// TIA Portal V20 export
TYPE "type_emRelations_em7_cmStatus"
// stored: Access Published, Namespace Unit1
   STRUCT
      cmSepaClampDetectSensor { ExternalAccessible := 'False'; ExternalVisible := 'False'; ExternalWritable := 'False'} : "LBC_typeDigitalSignalControlNode";
      cmSepaGripperDetectSensor { ExternalAccessible := 'False'; ExternalVisible := 'False'; ExternalWritable := 'False'} : "LBC_typeDigitalSignalControlNode";
      cmJRWinderDetectSensor { ExternalAccessible := 'False'; ExternalVisible := 'False'; ExternalWritable := 'False'} : "LBC_typeDigitalSignalControlNode";
      cmSepaClampSafetyPinDetectSensor { ExternalAccessible := 'False'; ExternalVisible := 'False'; ExternalWritable := 'False'} : "LBC_typeDigitalSignalControlNode";
      cmSepaGripperSafetyPinDetectSensor { ExternalAccessible := 'False'; ExternalVisible := 'False'; ExternalWritable := 'False'} : "LBC_typeDigitalSignalControlNode";
      cmSepaClampnCutterAxisX { ExternalAccessible := 'False'; ExternalVisible := 'False'; ExternalWritable := 'False'} : "LBC_typeAxis64PosControlNode";
      cmSepaClampnCutterAxisZ { ExternalAccessible := 'False'; ExternalVisible := 'False'; ExternalWritable := 'False'} : "LBC_typeAxis64PosControlNode";
      cmSepaGripperAxisX { ExternalAccessible := 'False'; ExternalVisible := 'False'; ExternalWritable := 'False'} : "LBC_typeAxis64PosControlNode";
      cmSepaGripperAxisZ { ExternalAccessible := 'False'; ExternalVisible := 'False'; ExternalWritable := 'False'} : "LBC_typeAxis64PosControlNode";
      cmSepaGripperAxisC { ExternalAccessible := 'False'; ExternalVisible := 'False'; ExternalWritable := 'False'} : "LBC_typeAxis64PosControlNode";
      cmJRWinderRearAxisY { ExternalAccessible := 'False'; ExternalVisible := 'False'; ExternalWritable := 'False'} : "LBC_typeAxis64PosControlNode";
      cmJRWinderFrontAxisY { ExternalAccessible := 'False'; ExternalVisible := 'False'; ExternalWritable := 'False'} : "LBC_typeAxis64PosControlNode";
      cmJRWinderAxisB { ExternalAccessible := 'False'; ExternalVisible := 'False'; ExternalWritable := 'False'} : "LBC_typeAxis64PosControlNode";
      cmJRPusherAxisZ { ExternalAccessible := 'False'; ExternalVisible := 'False'; ExternalWritable := 'False'} : "LBC_typeAxis64PosControlNode";
      cmSepaCutterUpDown { ExternalAccessible := 'False'; ExternalVisible := 'False'; ExternalWritable := 'False'} : "LBC_typeTwoWayActuatorControlNode";
      cmSepaClampTopUpDown { ExternalAccessible := 'False'; ExternalVisible := 'False'; ExternalWritable := 'False'} : "LBC_typeTwoWayActuatorControlNode";
      cmSepaClampBottomUpDown { ExternalAccessible := 'False'; ExternalVisible := 'False'; ExternalWritable := 'False'} : "LBC_typeTwoWayActuatorControlNode";
      cmStackGripperOpenClose { ExternalAccessible := 'False'; ExternalVisible := 'False'; ExternalWritable := 'False'} : "LBC_typeTwoWayActuatorControlNode";
      cmStackGripperFwdBwd { ExternalAccessible := 'False'; ExternalVisible := 'False'; ExternalWritable := 'False'} : "LBC_typeTwoWayActuatorControlNode";
      cmJRWinderClampTopRearUpDown { ExternalAccessible := 'False'; ExternalVisible := 'False'; ExternalWritable := 'False'} : "LBC_typeTwoWayActuatorControlNode";
      cmJRWinderClampBtmRearUpDown { ExternalAccessible := 'False'; ExternalVisible := 'False'; ExternalWritable := 'False'} : "LBC_typeTwoWayActuatorControlNode";
      cmJRWinderClampTopFrontUpDown { ExternalAccessible := 'False'; ExternalVisible := 'False'; ExternalWritable := 'False'} : "LBC_typeTwoWayActuatorControlNode";
      cmJRWinderClampBtmFrontUpDown { ExternalAccessible := 'False'; ExternalVisible := 'False'; ExternalWritable := 'False'} : "LBC_typeTwoWayActuatorControlNode";
      cmPusherRollerFwdBwd { ExternalAccessible := 'False'; ExternalVisible := 'False'; ExternalWritable := 'False'} : "LBC_typeTwoWayActuatorControlNode";
      cmHotWireCutter { ExternalAccessible := 'False'; ExternalVisible := 'False'; ExternalWritable := 'False'} : "LER_typeHotWireCutterControlNode";
   END_STRUCT;
   // cmSepaClampnCutterAxisX.commandConfiguration.power.startMode := 1;
   // cmSepaClampnCutterAxisX.commandConfiguration.power.stopMode := 0;
   // cmSepaClampnCutterAxisX.commandConfiguration.power.syncMotionSimulation := FALSE;
   // cmSepaClampnCutterAxisX.commandConfiguration.power.syncMotionSimulationExtendedMode := -1;
   // cmSepaClampnCutterAxisX.commandConfiguration.jog.velocity := 0.0;
   // cmSepaClampnCutterAxisX.commandConfiguration.jog.acceleration := -1.0;
   // cmSepaClampnCutterAxisX.commandConfiguration.jog.deceleration := -1.0;
   // cmSepaClampnCutterAxisX.commandConfiguration.jog.jerk := -1.0;
   // cmSepaClampnCutterAxisX.commandConfiguration.jog.positionControlled := TRUE;
   // cmSepaClampnCutterAxisX.commandConfiguration.jog.increment := 0.0;
   // cmSepaClampnCutterAxisX.commandConfiguration.jog.mode := 0;
   // cmSepaClampnCutterAxisX.commandConfiguration.moveVelocity.velocity := 0.0;
   // cmSepaClampnCutterAxisX.commandConfiguration.moveVelocity.acceleration := -1.0;
   // cmSepaClampnCutterAxisX.commandConfiguration.moveVelocity.deceleration := -1.0;
   // cmSepaClampnCutterAxisX.commandConfiguration.moveVelocity.jerk := -1.0;
   // cmSepaClampnCutterAxisX.commandConfiguration.moveVelocity.direction := 0;
   // cmSepaClampnCutterAxisX.commandConfiguration.moveVelocity.positionControlled := TRUE;
   // cmSepaClampnCutterAxisX.commandConfiguration.moveVelocity.velocityChangeOnTheFly := FALSE;
   // cmSepaClampnCutterAxisX.commandConfiguration.stop.deceleration := -1.0;
   // cmSepaClampnCutterAxisX.commandConfiguration.stop.jerk := -1.0;
   // cmSepaClampnCutterAxisX.commandConfiguration.stop.abortAcceleration := FALSE;
   // cmSepaClampnCutterAxisX.commandConfiguration.fastStop.deceleration := -1.0;
   // cmSepaClampnCutterAxisX.commandConfiguration.fastStop.jerk := -1.0;
   // cmSepaClampnCutterAxisX.commandConfiguration.fastStop.abortAcceleration := FALSE;
   // cmSepaClampnCutterAxisX.commandConfiguration.fastStop.replaceStopPossible := FALSE;
   // cmSepaClampnCutterAxisX.commandConfiguration.torqueLimiting.limit := -1.0;
   // cmSepaClampnCutterAxisX.commandConfiguration.torqueLimiting.mode := 0;
   // cmSepaClampnCutterAxisX.commandConfiguration.posRelative.distance := 0.0;
   // cmSepaClampnCutterAxisX.commandConfiguration.posRelative.velocity := -1.0;
   // cmSepaClampnCutterAxisX.commandConfiguration.posRelative.acceleration := -1.0;
   // cmSepaClampnCutterAxisX.commandConfiguration.posRelative.deceleration := -1.0;
   // cmSepaClampnCutterAxisX.commandConfiguration.posRelative.jerk := -1.0;
   // cmSepaClampnCutterAxisX.commandConfiguration.posRelative.direction := 0;
   // cmSepaClampnCutterAxisX.commandConfiguration.posAbsolute.position := 0.0;
   // cmSepaClampnCutterAxisX.commandConfiguration.posAbsolute.velocity := -1.0;
   // cmSepaClampnCutterAxisX.commandConfiguration.posAbsolute.acceleration := -1.0;
   // cmSepaClampnCutterAxisX.commandConfiguration.posAbsolute.deceleration := -1.0;
   // cmSepaClampnCutterAxisX.commandConfiguration.posAbsolute.jerk := -1.0;
   // cmSepaClampnCutterAxisX.commandConfiguration.posAbsolute.direction := 1;
   // cmSepaClampnCutterAxisX.commandConfiguration.posAbsolute.positionChangeOnTheFly := FALSE;
   // cmSepaClampnCutterAxisX.commandConfiguration.posAbsolute.velocityChangeOnTheFly := FALSE;
   // cmSepaClampnCutterAxisX.commandConfiguration.posSuperimposed.distance := 0.0;
   // cmSepaClampnCutterAxisX.commandConfiguration.posSuperimposed.velocityDiff := -1.0;
   // cmSepaClampnCutterAxisX.commandConfiguration.posSuperimposed.acceleration := -1.0;
   // cmSepaClampnCutterAxisX.commandConfiguration.posSuperimposed.deceleration := -1.0;
   // cmSepaClampnCutterAxisX.commandConfiguration.posSuperimposed.jerk := -1.0;
   // cmSepaClampnCutterAxisX.commandConfiguration.posSuperimposed.direction := 0;
   // cmSepaClampnCutterAxisX.commandConfiguration.haltSuperimposed.deceleration := -1.0;
   // cmSepaClampnCutterAxisX.commandConfiguration.haltSuperimposed.jerk := -1.0;
   // cmSepaClampnCutterAxisX.commandConfiguration.haltSuperimposed.abortAcceleration := FALSE;
   // cmSepaClampnCutterAxisX.commandConfiguration.gearInRelative.ratioNumerator := 1;
   // cmSepaClampnCutterAxisX.commandConfiguration.gearInRelative.ratioDenominator := 1;
   // cmSepaClampnCutterAxisX.commandConfiguration.gearInRelative.acceleration := -1.0;
   // cmSepaClampnCutterAxisX.commandConfiguration.gearInRelative.deceleration := -1.0;
   // cmSepaClampnCutterAxisX.commandConfiguration.gearInRelative.jerk := -1.0;
   // cmSepaClampnCutterAxisX.commandConfiguration.gearInRelative.ratioChangeOnTheFly := FALSE;
   // cmSepaClampnCutterAxisX.commandConfiguration.gearInAbsolute.ratioNumerator := 1;
   // cmSepaClampnCutterAxisX.commandConfiguration.gearInAbsolute.ratioDenominator := 1;
   // cmSepaClampnCutterAxisX.commandConfiguration.gearInAbsolute.masterSyncPosition := 0.0;
   // cmSepaClampnCutterAxisX.commandConfiguration.gearInAbsolute.slaveSyncPosition := 0.0;
   // cmSepaClampnCutterAxisX.commandConfiguration.gearInAbsolute.syncProfileReference := 1;
   // cmSepaClampnCutterAxisX.commandConfiguration.gearInAbsolute.masterStartDistance := 0.0;
   // cmSepaClampnCutterAxisX.commandConfiguration.gearInAbsolute.velocity := -1.0;
   // cmSepaClampnCutterAxisX.commandConfiguration.gearInAbsolute.acceleration := -1.0;
   // cmSepaClampnCutterAxisX.commandConfiguration.gearInAbsolute.deceleration := -1.0;
   // cmSepaClampnCutterAxisX.commandConfiguration.gearInAbsolute.jerk := -1.0;
   // cmSepaClampnCutterAxisX.commandConfiguration.gearInAbsolute.syncDirection := 1;
   // cmSepaClampnCutterAxisX.commandConfiguration.gearInAbsolute.ratioChangeOnTheFly := FALSE;
   // cmSepaClampnCutterAxisX.commandConfiguration.gearInVelocity.continuousUpdate := FALSE;
   // cmSepaClampnCutterAxisX.commandConfiguration.gearInVelocity.ratioNumerator := 1;
   // cmSepaClampnCutterAxisX.commandConfiguration.gearInVelocity.ratioDenominator := 1;
   // cmSepaClampnCutterAxisX.commandConfiguration.gearInVelocity.acceleration := -1.0;
   // cmSepaClampnCutterAxisX.commandConfiguration.gearInVelocity.deceleration := -1.0;
   // cmSepaClampnCutterAxisX.commandConfiguration.gearInVelocity.jerk := -1.0;
   // cmSepaClampnCutterAxisX.commandConfiguration.gearInVelocity.positionControlled := FALSE;
   // cmSepaClampnCutterAxisX.commandConfiguration.camIn.masterOffset := 0.0;
   // cmSepaClampnCutterAxisX.commandConfiguration.camIn.slaveOffset := 0.0;
   // cmSepaClampnCutterAxisX.commandConfiguration.camIn.masterScaling := 1.0;
   // cmSepaClampnCutterAxisX.commandConfiguration.camIn.slaveScaling := 1.0;
   // cmSepaClampnCutterAxisX.commandConfiguration.camIn.masterSyncPosition := 0.0;
   // cmSepaClampnCutterAxisX.commandConfiguration.camIn.syncProfileReference := 1;
   // cmSepaClampnCutterAxisX.commandConfiguration.camIn.masterStartDistance := 0.0;
   // cmSepaClampnCutterAxisX.commandConfiguration.camIn.velocity := -1.0;
   // cmSepaClampnCutterAxisX.commandConfiguration.camIn.acceleration := -1.0;
   // cmSepaClampnCutterAxisX.commandConfiguration.camIn.deceleration := -1.0;
   // cmSepaClampnCutterAxisX.commandConfiguration.camIn.jerk := -1.0;
   // cmSepaClampnCutterAxisX.commandConfiguration.camIn.applicationMode := 0;
   // cmSepaClampnCutterAxisX.commandConfiguration.camIn.syncDirection := 1;
   // cmSepaClampnCutterAxisX.commandConfiguration.gearOutCamOut.slavePosition := 0.0;
   // cmSepaClampnCutterAxisX.commandConfiguration.gearOutCamOut.syncProfileReference := 1;
   // cmSepaClampnCutterAxisX.commandConfiguration.gearOutCamOut.masterStopDistance := 0.0;
   // cmSepaClampnCutterAxisX.commandConfiguration.gearOutCamOut.deceleration := -1.0;
   // cmSepaClampnCutterAxisX.commandConfiguration.gearOutCamOut.jerk := -1.0;
   // cmSepaClampnCutterAxisX.commandConfiguration.gearOutCamOut.syncOutDirection := 3;
   // cmSepaClampnCutterAxisX.commandConfiguration.gearOutCamOut.gearOutCamOutMode := -1;
   // cmSepaClampnCutterAxisX.commandConfiguration.phasing.phaseShift := 0.0;
   // cmSepaClampnCutterAxisX.commandConfiguration.phasing.velocity := -1.0;
   // cmSepaClampnCutterAxisX.commandConfiguration.phasing.acceleration := -1.0;
   // cmSepaClampnCutterAxisX.commandConfiguration.phasing.deceleration := -1.0;
   // cmSepaClampnCutterAxisX.commandConfiguration.phasing.jerk := -1.0;
   // cmSepaClampnCutterAxisX.commandConfiguration.phasing.profileReference := 0;
   // cmSepaClampnCutterAxisX.commandConfiguration.phasing.phasingDistance := 0.0;
   // cmSepaClampnCutterAxisX.commandConfiguration.phasing.startPosition := 0.0;
   // cmSepaClampnCutterAxisX.commandConfiguration.phasing.direction := 3;
   // cmSepaClampnCutterAxisX.commandConfiguration.phasing.phaseAbsolute := TRUE;
   // cmSepaClampnCutterAxisX.commandConfiguration.phasing.phaseShiftChangeOnTheFly := FALSE;
   // cmSepaClampnCutterAxisX.commandConfiguration.offset.offset := 0.0;
   // cmSepaClampnCutterAxisX.commandConfiguration.offset.profileReference := 1;
   // cmSepaClampnCutterAxisX.commandConfiguration.offset.offsetDistance := 0.0;
   // cmSepaClampnCutterAxisX.commandConfiguration.offset.startPosition := 0.0;
   // cmSepaClampnCutterAxisX.commandConfiguration.offset.direction := 3;
   // cmSepaClampnCutterAxisX.commandConfiguration.offset.offsetAbsolute := TRUE;
   // cmSepaClampnCutterAxisX.commandConfiguration.offset.offsetChangeOnTheFly := FALSE;
   // cmSepaClampnCutterAxisZ.commandConfiguration.generalSettings.stopOnError := TRUE;
   // cmSepaClampnCutterAxisZ.commandConfiguration.generalSettings.resetWithRestart := FALSE;
   // cmSepaClampnCutterAxisZ.commandConfiguration.generalSettings.abortWaitingSyncCmd := TRUE;
   // cmSepaClampnCutterAxisZ.commandConfiguration.power.startMode := 1;
   // cmSepaClampnCutterAxisZ.commandConfiguration.power.stopMode := 0;
   // cmSepaClampnCutterAxisZ.commandConfiguration.power.syncMotionSimulation := FALSE;
   // cmSepaClampnCutterAxisZ.commandConfiguration.power.syncMotionSimulationExtendedMode := -1;
   // cmSepaClampnCutterAxisZ.commandConfiguration.jog.velocity := 0.0;
   // cmSepaClampnCutterAxisZ.commandConfiguration.jog.acceleration := -1.0;
   // cmSepaClampnCutterAxisZ.commandConfiguration.jog.deceleration := -1.0;
   // cmSepaClampnCutterAxisZ.commandConfiguration.jog.jerk := -1.0;
   // cmSepaClampnCutterAxisZ.commandConfiguration.jog.positionControlled := TRUE;
   // cmSepaClampnCutterAxisZ.commandConfiguration.jog.increment := 0.0;
   // cmSepaClampnCutterAxisZ.commandConfiguration.jog.mode := 0;
   // cmSepaClampnCutterAxisZ.commandConfiguration.moveVelocity.velocity := 0.0;
   // cmSepaClampnCutterAxisZ.commandConfiguration.moveVelocity.acceleration := -1.0;
   // cmSepaClampnCutterAxisZ.commandConfiguration.moveVelocity.deceleration := -1.0;
   // cmSepaClampnCutterAxisZ.commandConfiguration.moveVelocity.jerk := -1.0;
   // cmSepaClampnCutterAxisZ.commandConfiguration.moveVelocity.direction := 0;
   // cmSepaClampnCutterAxisZ.commandConfiguration.moveVelocity.positionControlled := TRUE;
   // cmSepaClampnCutterAxisZ.commandConfiguration.moveVelocity.velocityChangeOnTheFly := FALSE;
   // cmSepaClampnCutterAxisZ.commandConfiguration.stop.deceleration := -1.0;
   // cmSepaClampnCutterAxisZ.commandConfiguration.stop.jerk := -1.0;
   // cmSepaClampnCutterAxisZ.commandConfiguration.stop.abortAcceleration := FALSE;
   // cmSepaClampnCutterAxisZ.commandConfiguration.fastStop.deceleration := -1.0;
   // cmSepaClampnCutterAxisZ.commandConfiguration.fastStop.jerk := -1.0;
   // cmSepaClampnCutterAxisZ.commandConfiguration.fastStop.abortAcceleration := FALSE;
   // cmSepaClampnCutterAxisZ.commandConfiguration.fastStop.replaceStopPossible := FALSE;
   // cmSepaClampnCutterAxisZ.commandConfiguration.torqueLimiting.limit := -1.0;
   // cmSepaClampnCutterAxisZ.commandConfiguration.torqueLimiting.mode := 0;
   // cmSepaClampnCutterAxisZ.commandConfiguration.homing.position := 0.0;
   // cmSepaClampnCutterAxisZ.commandConfiguration.homing.mode := 0;
   // cmSepaClampnCutterAxisZ.commandConfiguration.homing.sensor := 0;
   // cmSepaClampnCutterAxisZ.commandConfiguration.homing.extendedMode := -1;
   // cmSepaClampnCutterAxisZ.commandConfiguration.homing.extendedModeTorqueLimit := 0.0;
   // cmSepaClampnCutterAxisZ.commandConfiguration.homing.extendedModeTargetPosition := 0.0;
   // cmSepaClampnCutterAxisZ.commandConfiguration.posRelative.distance := 0.0;
   // cmSepaClampnCutterAxisZ.commandConfiguration.posRelative.velocity := -1.0;
   // cmSepaClampnCutterAxisZ.commandConfiguration.posRelative.acceleration := -1.0;
   // cmSepaClampnCutterAxisZ.commandConfiguration.posRelative.deceleration := -1.0;
   // cmSepaClampnCutterAxisZ.commandConfiguration.posRelative.jerk := -1.0;
   // cmSepaClampnCutterAxisZ.commandConfiguration.posRelative.direction := 0;
   // cmSepaClampnCutterAxisZ.commandConfiguration.posAbsolute.position := 0.0;
   // cmSepaClampnCutterAxisZ.commandConfiguration.posAbsolute.velocity := -1.0;
   // cmSepaClampnCutterAxisZ.commandConfiguration.posAbsolute.acceleration := -1.0;
   // cmSepaClampnCutterAxisZ.commandConfiguration.posAbsolute.deceleration := -1.0;
   // cmSepaClampnCutterAxisZ.commandConfiguration.posAbsolute.jerk := -1.0;
   // cmSepaClampnCutterAxisZ.commandConfiguration.posAbsolute.direction := 1;
   // cmSepaClampnCutterAxisZ.commandConfiguration.posAbsolute.positionChangeOnTheFly := FALSE;
   // cmSepaClampnCutterAxisZ.commandConfiguration.posAbsolute.velocityChangeOnTheFly := FALSE;
   // cmSepaClampnCutterAxisZ.commandConfiguration.posSuperimposed.distance := 0.0;
   // cmSepaClampnCutterAxisZ.commandConfiguration.posSuperimposed.velocityDiff := -1.0;
   // cmSepaClampnCutterAxisZ.commandConfiguration.posSuperimposed.acceleration := -1.0;
   // cmSepaClampnCutterAxisZ.commandConfiguration.posSuperimposed.deceleration := -1.0;
   // cmSepaClampnCutterAxisZ.commandConfiguration.posSuperimposed.jerk := -1.0;
   // cmSepaClampnCutterAxisZ.commandConfiguration.posSuperimposed.direction := 0;
   // cmSepaClampnCutterAxisZ.commandConfiguration.haltSuperimposed.deceleration := -1.0;
   // cmSepaClampnCutterAxisZ.commandConfiguration.haltSuperimposed.jerk := -1.0;
   // cmSepaClampnCutterAxisZ.commandConfiguration.haltSuperimposed.abortAcceleration := FALSE;
   // cmSepaClampnCutterAxisZ.commandConfiguration.gearInRelative.ratioNumerator := 1;
   // cmSepaClampnCutterAxisZ.commandConfiguration.gearInRelative.ratioDenominator := 1;
   // cmSepaClampnCutterAxisZ.commandConfiguration.gearInRelative.acceleration := -1.0;
   // cmSepaClampnCutterAxisZ.commandConfiguration.gearInRelative.deceleration := -1.0;
   // cmSepaClampnCutterAxisZ.commandConfiguration.gearInRelative.jerk := -1.0;
   // cmSepaClampnCutterAxisZ.commandConfiguration.gearInRelative.ratioChangeOnTheFly := FALSE;
   // cmSepaClampnCutterAxisZ.commandConfiguration.gearInAbsolute.ratioNumerator := 1;
   // cmSepaClampnCutterAxisZ.commandConfiguration.gearInAbsolute.ratioDenominator := 1;
   // cmSepaClampnCutterAxisZ.commandConfiguration.gearInAbsolute.masterSyncPosition := 0.0;
   // cmSepaClampnCutterAxisZ.commandConfiguration.gearInAbsolute.slaveSyncPosition := 0.0;
   // cmSepaClampnCutterAxisZ.commandConfiguration.gearInAbsolute.syncProfileReference := 1;
   // cmSepaClampnCutterAxisZ.commandConfiguration.gearInAbsolute.masterStartDistance := 0.0;
   // cmSepaClampnCutterAxisZ.commandConfiguration.gearInAbsolute.velocity := -1.0;
   // cmSepaClampnCutterAxisZ.commandConfiguration.gearInAbsolute.acceleration := -1.0;
   // cmSepaClampnCutterAxisZ.commandConfiguration.gearInAbsolute.deceleration := -1.0;
   // cmSepaClampnCutterAxisZ.commandConfiguration.gearInAbsolute.jerk := -1.0;
   // cmSepaClampnCutterAxisZ.commandConfiguration.gearInAbsolute.syncDirection := 1;
   // cmSepaClampnCutterAxisZ.commandConfiguration.gearInAbsolute.ratioChangeOnTheFly := FALSE;
   // cmSepaClampnCutterAxisZ.commandConfiguration.gearInVelocity.continuousUpdate := FALSE;
   // cmSepaClampnCutterAxisZ.commandConfiguration.gearInVelocity.ratioNumerator := 1;
   // cmSepaClampnCutterAxisZ.commandConfiguration.gearInVelocity.ratioDenominator := 1;
   // cmSepaClampnCutterAxisZ.commandConfiguration.gearInVelocity.acceleration := -1.0;
   // cmSepaClampnCutterAxisZ.commandConfiguration.gearInVelocity.deceleration := -1.0;
   // cmSepaClampnCutterAxisZ.commandConfiguration.gearInVelocity.jerk := -1.0;
   // cmSepaClampnCutterAxisZ.commandConfiguration.gearInVelocity.positionControlled := FALSE;
   // cmSepaClampnCutterAxisZ.commandConfiguration.camIn.masterOffset := 0.0;
   // cmSepaClampnCutterAxisZ.commandConfiguration.camIn.slaveOffset := 0.0;
   // cmSepaClampnCutterAxisZ.commandConfiguration.camIn.masterScaling := 1.0;
   // cmSepaClampnCutterAxisZ.commandConfiguration.camIn.slaveScaling := 1.0;
   // cmSepaClampnCutterAxisZ.commandConfiguration.camIn.masterSyncPosition := 0.0;
   // cmSepaClampnCutterAxisZ.commandConfiguration.camIn.syncProfileReference := 1;
   // cmSepaClampnCutterAxisZ.commandConfiguration.camIn.masterStartDistance := 0.0;
   // cmSepaClampnCutterAxisZ.commandConfiguration.camIn.velocity := -1.0;
   // cmSepaClampnCutterAxisZ.commandConfiguration.camIn.acceleration := -1.0;
   // cmSepaClampnCutterAxisZ.commandConfiguration.camIn.deceleration := -1.0;
   // cmSepaClampnCutterAxisZ.commandConfiguration.camIn.jerk := -1.0;
   // cmSepaClampnCutterAxisZ.commandConfiguration.camIn.applicationMode := 0;
   // cmSepaClampnCutterAxisZ.commandConfiguration.camIn.syncDirection := 1;
   // cmSepaClampnCutterAxisZ.commandConfiguration.gearOutCamOut.slavePosition := 0.0;
   // cmSepaClampnCutterAxisZ.commandConfiguration.gearOutCamOut.syncProfileReference := 1;
   // cmSepaClampnCutterAxisZ.commandConfiguration.gearOutCamOut.masterStopDistance := 0.0;
   // cmSepaClampnCutterAxisZ.commandConfiguration.gearOutCamOut.deceleration := -1.0;
   // cmSepaClampnCutterAxisZ.commandConfiguration.gearOutCamOut.jerk := -1.0;
   // cmSepaClampnCutterAxisZ.commandConfiguration.gearOutCamOut.syncOutDirection := 3;
   // cmSepaClampnCutterAxisZ.commandConfiguration.gearOutCamOut.gearOutCamOutMode := -1;
   // cmSepaClampnCutterAxisZ.commandConfiguration.phasing.phaseShift := 0.0;
   // cmSepaClampnCutterAxisZ.commandConfiguration.phasing.velocity := -1.0;
   // cmSepaClampnCutterAxisZ.commandConfiguration.phasing.acceleration := -1.0;
   // cmSepaClampnCutterAxisZ.commandConfiguration.phasing.deceleration := -1.0;
   // cmSepaClampnCutterAxisZ.commandConfiguration.phasing.jerk := -1.0;
   // cmSepaClampnCutterAxisZ.commandConfiguration.phasing.profileReference := 0;
   // cmSepaClampnCutterAxisZ.commandConfiguration.phasing.phasingDistance := 0.0;
   // cmSepaClampnCutterAxisZ.commandConfiguration.phasing.startPosition := 0.0;
   // cmSepaClampnCutterAxisZ.commandConfiguration.phasing.direction := 3;
   // cmSepaClampnCutterAxisZ.commandConfiguration.phasing.phaseAbsolute := TRUE;
   // cmSepaClampnCutterAxisZ.commandConfiguration.phasing.phaseShiftChangeOnTheFly := FALSE;
   // cmSepaClampnCutterAxisZ.commandConfiguration.offset.offset := 0.0;
   // cmSepaClampnCutterAxisZ.commandConfiguration.offset.profileReference := 1;
   // cmSepaClampnCutterAxisZ.commandConfiguration.offset.offsetDistance := 0.0;
   // cmSepaClampnCutterAxisZ.commandConfiguration.offset.startPosition := 0.0;
   // cmSepaClampnCutterAxisZ.commandConfiguration.offset.direction := 3;
   // cmSepaClampnCutterAxisZ.commandConfiguration.offset.offsetAbsolute := TRUE;
   // cmSepaClampnCutterAxisZ.commandConfiguration.offset.offsetChangeOnTheFly := FALSE;
   // cmSepaClampnCutterAxisZ.commands.enableAxis := FALSE;
   // cmSepaClampnCutterAxisZ.commands.resetAxis := FALSE;
   // cmSepaClampnCutterAxisZ.commands.openBrake := FALSE;
   // cmSepaClampnCutterAxisZ.commands.jogForward := FALSE;
   // cmSepaClampnCutterAxisZ.commands.jogBackward := FALSE;
   // cmSepaClampnCutterAxisZ.commands.moveVelocity := FALSE;
   // cmSepaClampnCutterAxisZ.commands.stop := FALSE;
   // cmSepaClampnCutterAxisZ.commands.fastStop := FALSE;
   // cmSepaClampnCutterAxisZ.commands.torqueLimiting := FALSE;
   // cmSepaClampnCutterAxisZ.commands.homing := FALSE;
   // cmSepaClampnCutterAxisZ.commands.posRelative := FALSE;
   // cmSepaClampnCutterAxisZ.commands.posAbsolute := FALSE;
   // cmSepaClampnCutterAxisZ.commands.posSuperimposed := FALSE;
   // cmSepaClampnCutterAxisZ.commands.haltSuperimposed := FALSE;
   // cmSepaClampnCutterAxisZ.commands.selectSetPosition := -1;
   // cmSepaClampnCutterAxisZ.commands.reset := FALSE;
   // cmSepaGripperAxisX.commandConfiguration.stop.deceleration := -1.0;
   // cmSepaGripperAxisX.commandConfiguration.stop.jerk := -1.0;
   // cmSepaGripperAxisX.commandConfiguration.stop.abortAcceleration := FALSE;
   // cmSepaGripperAxisX.commandConfiguration.fastStop.deceleration := -1.0;
   // cmSepaGripperAxisX.commandConfiguration.fastStop.jerk := -1.0;
   // cmSepaGripperAxisX.commandConfiguration.fastStop.abortAcceleration := FALSE;
   // cmSepaGripperAxisX.commandConfiguration.fastStop.replaceStopPossible := FALSE;
   // cmSepaGripperAxisX.commandConfiguration.torqueLimiting.limit := -1.0;
   // cmSepaGripperAxisX.commandConfiguration.torqueLimiting.mode := 0;
   // cmSepaGripperAxisX.commandConfiguration.homing.position := 0.0;
   // cmSepaGripperAxisX.commandConfiguration.homing.mode := 0;
   // cmSepaGripperAxisX.commandConfiguration.homing.sensor := 0;
   // cmSepaGripperAxisX.commandConfiguration.homing.extendedMode := -1;
   // cmSepaGripperAxisX.commandConfiguration.homing.extendedModeTorqueLimit := 0.0;
   // cmSepaGripperAxisX.commandConfiguration.homing.extendedModeTargetPosition := 0.0;
   // cmSepaGripperAxisX.commandConfiguration.posRelative.distance := 0.0;
   // cmSepaGripperAxisX.commandConfiguration.posRelative.velocity := -1.0;
   // cmSepaGripperAxisX.commandConfiguration.posRelative.acceleration := -1.0;
   // cmSepaGripperAxisX.commandConfiguration.posRelative.deceleration := -1.0;
   // cmSepaGripperAxisX.commandConfiguration.posRelative.jerk := -1.0;
   // cmSepaGripperAxisX.commandConfiguration.posRelative.direction := 0;
   // cmSepaGripperAxisX.commandConfiguration.posAbsolute.position := 0.0;
   // cmSepaGripperAxisX.commandConfiguration.posAbsolute.velocity := -1.0;
   // cmSepaGripperAxisX.commandConfiguration.posAbsolute.acceleration := -1.0;
   // cmSepaGripperAxisX.commandConfiguration.posAbsolute.deceleration := -1.0;
   // cmSepaGripperAxisX.commandConfiguration.posAbsolute.jerk := -1.0;
   // cmSepaGripperAxisX.commandConfiguration.posAbsolute.direction := 1;
   // cmSepaGripperAxisX.commandConfiguration.posAbsolute.positionChangeOnTheFly := FALSE;
   // cmSepaGripperAxisX.commandConfiguration.posAbsolute.velocityChangeOnTheFly := FALSE;
   // cmSepaGripperAxisX.commandConfiguration.posSuperimposed.distance := 0.0;
   // cmSepaGripperAxisX.commandConfiguration.posSuperimposed.velocityDiff := -1.0;
   // cmSepaGripperAxisX.commandConfiguration.posSuperimposed.acceleration := -1.0;
   // cmSepaGripperAxisX.commandConfiguration.posSuperimposed.deceleration := -1.0;
   // cmSepaGripperAxisX.commandConfiguration.posSuperimposed.jerk := -1.0;
   // cmSepaGripperAxisX.commandConfiguration.posSuperimposed.direction := 0;
   // cmSepaGripperAxisX.commandConfiguration.haltSuperimposed.deceleration := -1.0;
   // cmSepaGripperAxisX.commandConfiguration.haltSuperimposed.jerk := -1.0;
   // cmSepaGripperAxisX.commandConfiguration.haltSuperimposed.abortAcceleration := FALSE;
   // cmSepaGripperAxisX.commandConfiguration.gearInRelative.ratioNumerator := 1;
   // cmSepaGripperAxisX.commandConfiguration.gearInRelative.ratioDenominator := 1;
   // cmSepaGripperAxisX.commandConfiguration.gearInRelative.acceleration := -1.0;
   // cmSepaGripperAxisX.commandConfiguration.gearInRelative.deceleration := -1.0;
   // cmSepaGripperAxisX.commandConfiguration.gearInRelative.jerk := -1.0;
   // cmSepaGripperAxisX.commandConfiguration.gearInRelative.ratioChangeOnTheFly := FALSE;
   // cmSepaGripperAxisX.commandConfiguration.gearInAbsolute.ratioNumerator := 1;
   // cmSepaGripperAxisX.commandConfiguration.gearInAbsolute.ratioDenominator := 1;
   // cmSepaGripperAxisX.commandConfiguration.gearInAbsolute.masterSyncPosition := 0.0;
   // cmSepaGripperAxisX.commandConfiguration.gearInAbsolute.slaveSyncPosition := 0.0;
   // cmSepaGripperAxisX.commandConfiguration.gearInAbsolute.syncProfileReference := 1;
   // cmSepaGripperAxisX.commandConfiguration.gearInAbsolute.masterStartDistance := 0.0;
   // cmSepaGripperAxisX.commandConfiguration.gearInAbsolute.velocity := -1.0;
   // cmSepaGripperAxisX.commandConfiguration.gearInAbsolute.acceleration := -1.0;
   // cmSepaGripperAxisX.commandConfiguration.gearInAbsolute.deceleration := -1.0;
   // cmSepaGripperAxisX.commandConfiguration.gearInAbsolute.jerk := -1.0;
   // cmSepaGripperAxisX.commandConfiguration.gearInAbsolute.syncDirection := 1;
   // cmSepaGripperAxisX.commandConfiguration.gearInAbsolute.ratioChangeOnTheFly := FALSE;
   // cmSepaGripperAxisX.commandConfiguration.gearInVelocity.continuousUpdate := FALSE;
   // cmSepaGripperAxisX.commandConfiguration.gearInVelocity.ratioNumerator := 1;
   // cmSepaGripperAxisX.commandConfiguration.gearInVelocity.ratioDenominator := 1;
   // cmSepaGripperAxisX.commandConfiguration.gearInVelocity.acceleration := -1.0;
   // cmSepaGripperAxisX.commandConfiguration.gearInVelocity.deceleration := -1.0;
   // cmSepaGripperAxisX.commandConfiguration.gearInVelocity.jerk := -1.0;
   // cmSepaGripperAxisX.commandConfiguration.gearInVelocity.positionControlled := FALSE;
   // cmSepaGripperAxisX.commandConfiguration.camIn.masterOffset := 0.0;
   // cmSepaGripperAxisX.commandConfiguration.camIn.slaveOffset := 0.0;
   // cmSepaGripperAxisX.commandConfiguration.camIn.masterScaling := 1.0;
   // cmSepaGripperAxisX.commandConfiguration.camIn.slaveScaling := 1.0;
   // cmSepaGripperAxisX.commandConfiguration.camIn.masterSyncPosition := 0.0;
   // cmSepaGripperAxisX.commandConfiguration.camIn.syncProfileReference := 1;
   // cmSepaGripperAxisX.commandConfiguration.camIn.masterStartDistance := 0.0;
   // cmSepaGripperAxisX.commandConfiguration.camIn.velocity := -1.0;
   // cmSepaGripperAxisX.commandConfiguration.camIn.acceleration := -1.0;
   // cmSepaGripperAxisX.commandConfiguration.camIn.deceleration := -1.0;
   // cmSepaGripperAxisX.commandConfiguration.camIn.jerk := -1.0;
   // cmSepaGripperAxisX.commandConfiguration.camIn.applicationMode := 0;
   // cmSepaGripperAxisX.commandConfiguration.camIn.syncDirection := 1;
   // cmSepaGripperAxisX.commandConfiguration.gearOutCamOut.slavePosition := 0.0;
   // cmSepaGripperAxisX.commandConfiguration.gearOutCamOut.syncProfileReference := 1;
   // cmSepaGripperAxisX.commandConfiguration.gearOutCamOut.masterStopDistance := 0.0;
   // cmSepaGripperAxisX.commandConfiguration.gearOutCamOut.deceleration := -1.0;
   // cmSepaGripperAxisX.commandConfiguration.gearOutCamOut.jerk := -1.0;
   // cmSepaGripperAxisX.commandConfiguration.gearOutCamOut.syncOutDirection := 3;
   // cmSepaGripperAxisX.commandConfiguration.gearOutCamOut.gearOutCamOutMode := -1;
   // cmSepaGripperAxisX.commandConfiguration.phasing.phaseShift := 0.0;
   // cmSepaGripperAxisX.commandConfiguration.phasing.velocity := -1.0;
   // cmSepaGripperAxisX.commandConfiguration.phasing.acceleration := -1.0;
   // cmSepaGripperAxisX.commandConfiguration.phasing.deceleration := -1.0;
   // cmSepaGripperAxisX.commandConfiguration.phasing.jerk := -1.0;
   // cmSepaGripperAxisX.commandConfiguration.phasing.profileReference := 0;
   // cmSepaGripperAxisX.commandConfiguration.phasing.phasingDistance := 0.0;
   // cmSepaGripperAxisX.commandConfiguration.phasing.startPosition := 0.0;
   // cmSepaGripperAxisX.commandConfiguration.phasing.direction := 3;
   // cmSepaGripperAxisX.commandConfiguration.phasing.phaseAbsolute := TRUE;
   // cmSepaGripperAxisX.commandConfiguration.phasing.phaseShiftChangeOnTheFly := FALSE;
   // cmSepaGripperAxisX.commandConfiguration.offset.offset := 0.0;
   // cmSepaGripperAxisX.commandConfiguration.offset.profileReference := 1;
   // cmSepaGripperAxisX.commandConfiguration.offset.offsetDistance := 0.0;
   // cmSepaGripperAxisX.commandConfiguration.offset.startPosition := 0.0;
   // cmSepaGripperAxisX.commandConfiguration.offset.direction := 3;
   // cmSepaGripperAxisX.commandConfiguration.offset.offsetAbsolute := TRUE;
   // cmSepaGripperAxisX.commandConfiguration.offset.offsetChangeOnTheFly := FALSE;
   // cmSepaGripperAxisZ.commandConfiguration.generalSettings.stopOnError := TRUE;
   // cmSepaGripperAxisZ.commandConfiguration.generalSettings.resetWithRestart := FALSE;
   // cmSepaGripperAxisZ.commandConfiguration.generalSettings.abortWaitingSyncCmd := TRUE;
   // cmSepaGripperAxisZ.commandConfiguration.power.startMode := 1;
   // cmSepaGripperAxisZ.commandConfiguration.power.stopMode := 0;
   // cmSepaGripperAxisZ.commandConfiguration.power.syncMotionSimulation := FALSE;
   // cmSepaGripperAxisZ.commandConfiguration.power.syncMotionSimulationExtendedMode := -1;
   // cmSepaGripperAxisZ.commandConfiguration.jog.velocity := 0.0;
   // cmSepaGripperAxisZ.commandConfiguration.jog.acceleration := -1.0;
   // cmSepaGripperAxisZ.commandConfiguration.jog.deceleration := -1.0;
   // cmSepaGripperAxisZ.commandConfiguration.jog.jerk := -1.0;
   // cmSepaGripperAxisZ.commandConfiguration.jog.positionControlled := TRUE;
   // cmSepaGripperAxisZ.commandConfiguration.jog.increment := 0.0;
   // cmSepaGripperAxisZ.commandConfiguration.jog.mode := 0;
   // cmSepaGripperAxisZ.commandConfiguration.moveVelocity.velocity := 0.0;
   // cmSepaGripperAxisZ.commandConfiguration.moveVelocity.acceleration := -1.0;
   // cmSepaGripperAxisZ.commandConfiguration.moveVelocity.deceleration := -1.0;
   // cmSepaGripperAxisZ.commandConfiguration.moveVelocity.jerk := -1.0;
   // cmSepaGripperAxisZ.commandConfiguration.moveVelocity.direction := 0;
   // cmSepaGripperAxisZ.commandConfiguration.moveVelocity.positionControlled := TRUE;
   // cmSepaGripperAxisZ.commandConfiguration.moveVelocity.velocityChangeOnTheFly := FALSE;
   // cmSepaGripperAxisZ.commandConfiguration.stop.deceleration := -1.0;
   // cmSepaGripperAxisZ.commandConfiguration.stop.jerk := -1.0;
   // cmSepaGripperAxisZ.commandConfiguration.stop.abortAcceleration := FALSE;
   // cmSepaGripperAxisZ.commandConfiguration.fastStop.deceleration := -1.0;
   // cmSepaGripperAxisZ.commandConfiguration.fastStop.jerk := -1.0;
   // cmSepaGripperAxisZ.commandConfiguration.fastStop.abortAcceleration := FALSE;
   // cmSepaGripperAxisZ.commandConfiguration.fastStop.replaceStopPossible := FALSE;
   // cmSepaGripperAxisZ.commandConfiguration.torqueLimiting.limit := -1.0;
   // cmSepaGripperAxisZ.commandConfiguration.torqueLimiting.mode := 0;
   // cmSepaGripperAxisZ.commandConfiguration.homing.position := 0.0;
   // cmSepaGripperAxisZ.commandConfiguration.homing.mode := 0;
   // cmSepaGripperAxisZ.commandConfiguration.homing.sensor := 0;
   // cmSepaGripperAxisZ.commandConfiguration.homing.extendedMode := -1;
   // cmSepaGripperAxisZ.commandConfiguration.homing.extendedModeTorqueLimit := 0.0;
   // cmSepaGripperAxisZ.commandConfiguration.homing.extendedModeTargetPosition := 0.0;
   // cmSepaGripperAxisZ.commandConfiguration.posRelative.distance := 0.0;
   // cmSepaGripperAxisZ.commandConfiguration.posRelative.velocity := -1.0;
   // cmSepaGripperAxisZ.commandConfiguration.posRelative.acceleration := -1.0;
   // cmSepaGripperAxisZ.commandConfiguration.posRelative.deceleration := -1.0;
   // cmSepaGripperAxisZ.commandConfiguration.posRelative.jerk := -1.0;
   // cmSepaGripperAxisZ.commandConfiguration.posRelative.direction := 0;
   // cmSepaGripperAxisZ.commandConfiguration.posAbsolute.position := 0.0;
   // cmSepaGripperAxisZ.commandConfiguration.posAbsolute.velocity := -1.0;
   // cmSepaGripperAxisZ.commandConfiguration.posAbsolute.acceleration := -1.0;
   // cmSepaGripperAxisZ.commandConfiguration.posAbsolute.deceleration := -1.0;
   // cmSepaGripperAxisZ.commandConfiguration.posAbsolute.jerk := -1.0;
   // cmSepaGripperAxisZ.commandConfiguration.posAbsolute.direction := 1;
   // cmSepaGripperAxisZ.commandConfiguration.posAbsolute.positionChangeOnTheFly := FALSE;
   // cmSepaGripperAxisZ.commandConfiguration.posAbsolute.velocityChangeOnTheFly := FALSE;
   // cmSepaGripperAxisZ.commandConfiguration.posSuperimposed.distance := 0.0;
   // cmSepaGripperAxisZ.commandConfiguration.posSuperimposed.velocityDiff := -1.0;
   // cmSepaGripperAxisZ.commandConfiguration.posSuperimposed.acceleration := -1.0;
   // cmSepaGripperAxisZ.commandConfiguration.posSuperimposed.deceleration := -1.0;
   // cmSepaGripperAxisZ.commandConfiguration.posSuperimposed.jerk := -1.0;
   // cmSepaGripperAxisZ.commandConfiguration.posSuperimposed.direction := 0;
   // cmSepaGripperAxisZ.commandConfiguration.haltSuperimposed.deceleration := -1.0;
   // cmSepaGripperAxisZ.commandConfiguration.haltSuperimposed.jerk := -1.0;
   // cmSepaGripperAxisZ.commandConfiguration.haltSuperimposed.abortAcceleration := FALSE;
   // cmSepaGripperAxisZ.commandConfiguration.gearInRelative.ratioNumerator := 1;
   // cmSepaGripperAxisZ.commandConfiguration.gearInRelative.ratioDenominator := 1;
   // cmSepaGripperAxisZ.commandConfiguration.gearInRelative.acceleration := -1.0;
   // cmSepaGripperAxisZ.commandConfiguration.gearInRelative.deceleration := -1.0;
   // cmSepaGripperAxisZ.commandConfiguration.gearInRelative.jerk := -1.0;
   // cmSepaGripperAxisZ.commandConfiguration.gearInRelative.ratioChangeOnTheFly := FALSE;
   // cmSepaGripperAxisZ.commandConfiguration.gearInAbsolute.ratioNumerator := 1;
   // cmSepaGripperAxisZ.commandConfiguration.gearInAbsolute.ratioDenominator := 1;
   // cmSepaGripperAxisZ.commandConfiguration.gearInAbsolute.masterSyncPosition := 0.0;
   // cmSepaGripperAxisZ.commandConfiguration.gearInAbsolute.slaveSyncPosition := 0.0;
   // cmSepaGripperAxisZ.commandConfiguration.gearInAbsolute.syncProfileReference := 1;
   // cmSepaGripperAxisZ.commandConfiguration.gearInAbsolute.masterStartDistance := 0.0;
   // cmSepaGripperAxisZ.commandConfiguration.gearInAbsolute.velocity := -1.0;
   // cmSepaGripperAxisZ.commandConfiguration.gearInAbsolute.acceleration := -1.0;
   // cmSepaGripperAxisZ.commandConfiguration.gearInAbsolute.deceleration := -1.0;
   // cmSepaGripperAxisZ.commandConfiguration.gearInAbsolute.jerk := -1.0;
   // cmSepaGripperAxisZ.commandConfiguration.gearInAbsolute.syncDirection := 1;
   // cmSepaGripperAxisZ.commandConfiguration.gearInAbsolute.ratioChangeOnTheFly := FALSE;
   // cmSepaGripperAxisZ.commandConfiguration.gearInVelocity.continuousUpdate := FALSE;
   // cmSepaGripperAxisZ.commandConfiguration.gearInVelocity.ratioNumerator := 1;
   // cmSepaGripperAxisZ.commandConfiguration.gearInVelocity.ratioDenominator := 1;
   // cmSepaGripperAxisZ.commandConfiguration.gearInVelocity.acceleration := -1.0;
   // cmSepaGripperAxisZ.commandConfiguration.gearInVelocity.deceleration := -1.0;
   // cmSepaGripperAxisZ.commandConfiguration.gearInVelocity.jerk := -1.0;
   // cmSepaGripperAxisZ.commandConfiguration.gearInVelocity.positionControlled := FALSE;
   // cmSepaGripperAxisZ.commandConfiguration.camIn.masterOffset := 0.0;
   // cmSepaGripperAxisZ.commandConfiguration.camIn.slaveOffset := 0.0;
   // cmSepaGripperAxisZ.commandConfiguration.camIn.masterScaling := 1.0;
   // cmSepaGripperAxisZ.commandConfiguration.camIn.slaveScaling := 1.0;
   // cmSepaGripperAxisZ.commandConfiguration.camIn.masterSyncPosition := 0.0;
   // cmSepaGripperAxisZ.commandConfiguration.camIn.syncProfileReference := 1;
   // cmSepaGripperAxisZ.commandConfiguration.camIn.masterStartDistance := 0.0;
   // cmSepaGripperAxisZ.commandConfiguration.camIn.velocity := -1.0;
   // cmSepaGripperAxisZ.commandConfiguration.camIn.acceleration := -1.0;
   // cmSepaGripperAxisZ.commandConfiguration.camIn.deceleration := -1.0;
   // cmSepaGripperAxisZ.commandConfiguration.camIn.jerk := -1.0;
   // cmSepaGripperAxisZ.commandConfiguration.camIn.applicationMode := 0;
   // cmSepaGripperAxisZ.commandConfiguration.camIn.syncDirection := 1;
   // cmSepaGripperAxisZ.commandConfiguration.gearOutCamOut.slavePosition := 0.0;
   // cmSepaGripperAxisZ.commandConfiguration.gearOutCamOut.syncProfileReference := 1;
   // cmSepaGripperAxisZ.commandConfiguration.gearOutCamOut.masterStopDistance := 0.0;
   // cmSepaGripperAxisZ.commandConfiguration.gearOutCamOut.deceleration := -1.0;
   // cmSepaGripperAxisZ.commandConfiguration.gearOutCamOut.jerk := -1.0;
   // cmSepaGripperAxisZ.commandConfiguration.gearOutCamOut.syncOutDirection := 3;
   // cmSepaGripperAxisZ.commandConfiguration.gearOutCamOut.gearOutCamOutMode := -1;
   // cmSepaGripperAxisZ.commandConfiguration.phasing.phaseShift := 0.0;
   // cmSepaGripperAxisZ.commandConfiguration.phasing.velocity := -1.0;
   // cmSepaGripperAxisZ.commandConfiguration.phasing.acceleration := -1.0;
   // cmSepaGripperAxisZ.commandConfiguration.phasing.deceleration := -1.0;
   // cmSepaGripperAxisZ.commandConfiguration.phasing.jerk := -1.0;
   // cmSepaGripperAxisZ.commandConfiguration.phasing.profileReference := 0;
   // cmSepaGripperAxisZ.commandConfiguration.phasing.phasingDistance := 0.0;
   // cmSepaGripperAxisZ.commandConfiguration.phasing.startPosition := 0.0;
   // cmSepaGripperAxisZ.commandConfiguration.phasing.direction := 3;
   // cmSepaGripperAxisZ.commandConfiguration.phasing.phaseAbsolute := TRUE;
   // cmSepaGripperAxisZ.commandConfiguration.phasing.phaseShiftChangeOnTheFly := FALSE;
   // cmSepaGripperAxisZ.commandConfiguration.offset.offset := 0.0;
   // cmSepaGripperAxisZ.commandConfiguration.offset.profileReference := 1;
   // cmSepaGripperAxisZ.commandConfiguration.offset.offsetDistance := 0.0;
   // cmSepaGripperAxisZ.commandConfiguration.offset.startPosition := 0.0;
   // cmSepaGripperAxisZ.commandConfiguration.offset.direction := 3;
   // cmSepaGripperAxisZ.commandConfiguration.offset.offsetAbsolute := TRUE;
   // cmSepaGripperAxisZ.commandConfiguration.offset.offsetChangeOnTheFly := FALSE;
   // cmSepaGripperAxisZ.commands.enableAxis := FALSE;
   // cmSepaGripperAxisZ.commands.resetAxis := FALSE;
   // cmSepaGripperAxisZ.commands.openBrake := FALSE;
   // cmSepaGripperAxisZ.commands.jogForward := FALSE;
   // cmSepaGripperAxisZ.commands.jogBackward := FALSE;
   // cmSepaGripperAxisZ.commands.moveVelocity := FALSE;
   // cmSepaGripperAxisZ.commands.stop := FALSE;
   // cmSepaGripperAxisZ.commands.fastStop := FALSE;
   // cmSepaGripperAxisZ.commands.torqueLimiting := FALSE;
   // cmSepaGripperAxisZ.commands.homing := FALSE;
   // cmSepaGripperAxisZ.commands.posRelative := FALSE;
   // cmSepaGripperAxisZ.commands.posAbsolute := FALSE;
   // cmSepaGripperAxisZ.commands.posSuperimposed := FALSE;
   // cmSepaGripperAxisZ.commands.haltSuperimposed := FALSE;
   // cmSepaGripperAxisZ.commands.selectSetPosition := -1;
   // cmSepaGripperAxisZ.commands.reset := FALSE;
   // cmSepaGripperAxisZ.monitoring.valid := FALSE;
   // cmSepaGripperAxisZ.monitoring.busy := TRUE;
   // cmSepaGripperAxisZ.monitoring.error := TRUE;
   // cmSepaGripperAxisZ.monitoring.status := 16#8600;
   // cmSepaGripperAxisZ.monitoring.subfunctionStatus := 16#8001;
   // cmSepaGripperAxisZ.monitoring.axisEnabled := FALSE;
   // cmSepaGripperAxisZ.monitoring.resetActive := FALSE;
   // cmSepaGripperAxisZ.monitoring.inVelocity := FALSE;
   // cmSepaGripperAxisZ.monitoring.inLimitation := FALSE;
   // cmSepaGripperAxisZ.monitoring.inClamping := FALSE;
   // cmSepaGripperAxisZ.monitoring.startSync := FALSE;
   // cmSepaGripperAxisZ.monitoring.inSync := FALSE;
   // cmSepaGripperAxisZ.monitoring.inSimulation := FALSE;
   // cmSepaGripperAxisZ.monitoring.jogSelected := FALSE;
   // cmSepaGripperAxisZ.monitoring.moveVelocitySelected := FALSE;
   // cmSepaGripperAxisZ.monitoring.stopSelected := FALSE;
   // cmSepaGripperAxisZ.monitoring.fastStopSelected := FALSE;
   // cmSepaGripperAxisZ.monitoring.torqueLimitingSelected := FALSE;
   // cmSepaGripperAxisZ.monitoring.homingSelected := FALSE;
   // cmSepaGripperAxisZ.monitoring.posRelativeSelected := FALSE;
   // cmSepaGripperAxisZ.monitoring.posAbsoluteSelected := FALSE;
   // cmSepaGripperAxisZ.monitoring.posSuperimposedSelected := FALSE;
   // cmSepaGripperAxisZ.monitoring.haltSuperimposedSelected := FALSE;
   // cmSepaGripperAxisZ.monitoring.commandBusy := FALSE;
   // cmSepaGripperAxisZ.monitoring.commandDone := FALSE;
   // cmSepaGripperAxisZ.monitoring.commandAborted := FALSE;
   // cmSepaGripperAxisZ.monitoring.homingCommandBusy := FALSE;
   // cmSepaGripperAxisZ.monitoring.homingCommandDone := FALSE;
   // cmSepaGripperAxisZ.monitoring.homingCommandAborted := FALSE;
   // cmSepaGripperAxisZ.monitoring.superimposedBusy := FALSE;
   // cmSepaGripperAxisZ.monitoring.superimposedDone := FALSE;
   // cmSepaGripperAxisZ.monitoring.superimposedAborted := FALSE;
   // cmSepaGripperAxisZ.monitoring.actualPosition := 159.839;
   // cmSepaGripperAxisZ.monitoring.actualSpeed := 0.0;
   // cmSepaGripperAxisZ.monitoring.speedUnit := 1062;
   // cmSepaGripperAxisZ.monitoring.positionUnit := 1013;
   // cmSepaGripperAxisZ.monitoring.axisType := 1;
   // cmSepaGripperAxisZ.monitoring.interlockGeneralOut := TRUE;
   // cmSepaGripperAxisZ.monitoring.interlockJogForwardOut := TRUE;
   // cmSepaGripperAxisZ.monitoring.interlockJogBackwardOut := TRUE;
   // cmSepaGripperAxisC.commandConfiguration.generalSettings.stopOnError := TRUE;
   // cmSepaGripperAxisC.commandConfiguration.generalSettings.resetWithRestart := FALSE;
   // cmSepaGripperAxisC.commandConfiguration.generalSettings.abortWaitingSyncCmd := TRUE;
   // cmSepaGripperAxisC.commandConfiguration.power.startMode := 1;
   // cmSepaGripperAxisC.commandConfiguration.power.stopMode := 0;
   // cmSepaGripperAxisC.commandConfiguration.power.syncMotionSimulation := FALSE;
   // cmSepaGripperAxisC.commandConfiguration.power.syncMotionSimulationExtendedMode := -1;
   // cmSepaGripperAxisC.commandConfiguration.jog.velocity := 0.0;
   // cmSepaGripperAxisC.commandConfiguration.jog.acceleration := -1.0;
   // cmSepaGripperAxisC.commandConfiguration.jog.deceleration := -1.0;
   // cmSepaGripperAxisC.commandConfiguration.jog.jerk := -1.0;
   // cmSepaGripperAxisC.commandConfiguration.jog.positionControlled := TRUE;
   // cmSepaGripperAxisC.commandConfiguration.jog.increment := 0.0;
   // cmSepaGripperAxisC.commandConfiguration.jog.mode := 0;
   // cmSepaGripperAxisC.commandConfiguration.moveVelocity.velocity := 0.0;
   // cmSepaGripperAxisC.commandConfiguration.moveVelocity.acceleration := -1.0;
   // cmSepaGripperAxisC.commandConfiguration.moveVelocity.deceleration := -1.0;
   // cmSepaGripperAxisC.commandConfiguration.moveVelocity.jerk := -1.0;
   // cmSepaGripperAxisC.commandConfiguration.moveVelocity.direction := 0;
   // cmSepaGripperAxisC.commandConfiguration.moveVelocity.positionControlled := TRUE;
   // cmSepaGripperAxisC.commandConfiguration.moveVelocity.velocityChangeOnTheFly := FALSE;
   // cmSepaGripperAxisC.commandConfiguration.stop.deceleration := -1.0;
   // cmSepaGripperAxisC.commandConfiguration.stop.jerk := -1.0;
   // cmSepaGripperAxisC.commandConfiguration.stop.abortAcceleration := FALSE;
   // cmSepaGripperAxisC.commandConfiguration.fastStop.deceleration := -1.0;
   // cmSepaGripperAxisC.commandConfiguration.fastStop.jerk := -1.0;
   // cmSepaGripperAxisC.commandConfiguration.fastStop.abortAcceleration := FALSE;
   // cmSepaGripperAxisC.commandConfiguration.fastStop.replaceStopPossible := FALSE;
   // cmSepaGripperAxisC.commandConfiguration.torqueLimiting.limit := -1.0;
   // cmSepaGripperAxisC.commandConfiguration.torqueLimiting.mode := 0;
   // cmSepaGripperAxisC.commandConfiguration.homing.position := 0.0;
   // cmSepaGripperAxisC.commandConfiguration.homing.mode := 0;
   // cmSepaGripperAxisC.commandConfiguration.homing.sensor := 0;
   // cmSepaGripperAxisC.commandConfiguration.homing.extendedMode := -1;
   // cmSepaGripperAxisC.commandConfiguration.homing.extendedModeTorqueLimit := 0.0;
   // cmSepaGripperAxisC.commandConfiguration.homing.extendedModeTargetPosition := 0.0;
   // cmSepaGripperAxisC.commandConfiguration.posRelative.distance := 0.0;
   // cmSepaGripperAxisC.commandConfiguration.posRelative.velocity := -1.0;
   // cmSepaGripperAxisC.commandConfiguration.posRelative.acceleration := -1.0;
   // cmSepaGripperAxisC.commandConfiguration.posRelative.deceleration := -1.0;
   // cmSepaGripperAxisC.commandConfiguration.posRelative.jerk := -1.0;
   // cmSepaGripperAxisC.commandConfiguration.posRelative.direction := 0;
   // cmSepaGripperAxisC.commandConfiguration.posAbsolute.position := 0.0;
   // cmSepaGripperAxisC.commandConfiguration.posAbsolute.velocity := -1.0;
   // cmSepaGripperAxisC.commandConfiguration.posAbsolute.acceleration := -1.0;
   // cmSepaGripperAxisC.commandConfiguration.posAbsolute.deceleration := -1.0;
   // cmSepaGripperAxisC.commandConfiguration.posAbsolute.jerk := -1.0;
   // cmSepaGripperAxisC.commandConfiguration.posAbsolute.direction := 1;
   // cmSepaGripperAxisC.commandConfiguration.posAbsolute.positionChangeOnTheFly := FALSE;
   // cmSepaGripperAxisC.commandConfiguration.posAbsolute.velocityChangeOnTheFly := FALSE;
   // cmSepaGripperAxisC.commandConfiguration.posSuperimposed.distance := 0.0;
   // cmSepaGripperAxisC.commandConfiguration.posSuperimposed.velocityDiff := -1.0;
   // cmSepaGripperAxisC.commandConfiguration.posSuperimposed.acceleration := -1.0;
   // cmSepaGripperAxisC.commandConfiguration.posSuperimposed.deceleration := -1.0;
   // cmSepaGripperAxisC.commandConfiguration.posSuperimposed.jerk := -1.0;
   // cmSepaGripperAxisC.commandConfiguration.posSuperimposed.direction := 0;
   // cmSepaGripperAxisC.commandConfiguration.haltSuperimposed.deceleration := -1.0;
   // cmSepaGripperAxisC.commandConfiguration.haltSuperimposed.jerk := -1.0;
   // cmSepaGripperAxisC.commandConfiguration.haltSuperimposed.abortAcceleration := FALSE;
   // cmSepaGripperAxisC.commandConfiguration.gearInRelative.ratioNumerator := 1;
   // cmSepaGripperAxisC.commandConfiguration.gearInRelative.ratioDenominator := 1;
   // cmSepaGripperAxisC.commandConfiguration.gearInRelative.acceleration := -1.0;
   // cmSepaGripperAxisC.commandConfiguration.gearInRelative.deceleration := -1.0;
   // cmSepaGripperAxisC.commandConfiguration.gearInRelative.jerk := -1.0;
   // cmSepaGripperAxisC.commandConfiguration.gearInRelative.ratioChangeOnTheFly := FALSE;
   // cmSepaGripperAxisC.commandConfiguration.gearInAbsolute.ratioNumerator := 1;
   // cmSepaGripperAxisC.commandConfiguration.gearInAbsolute.ratioDenominator := 1;
   // cmSepaGripperAxisC.commandConfiguration.gearInAbsolute.masterSyncPosition := 0.0;
   // cmSepaGripperAxisC.commandConfiguration.gearInAbsolute.slaveSyncPosition := 0.0;
   // cmSepaGripperAxisC.commandConfiguration.gearInAbsolute.syncProfileReference := 1;
   // cmSepaGripperAxisC.commandConfiguration.gearInAbsolute.masterStartDistance := 0.0;
   // cmSepaGripperAxisC.commandConfiguration.gearInAbsolute.velocity := -1.0;
   // cmSepaGripperAxisC.commandConfiguration.gearInAbsolute.acceleration := -1.0;
   // cmSepaGripperAxisC.commandConfiguration.gearInAbsolute.deceleration := -1.0;
   // cmSepaGripperAxisC.commandConfiguration.gearInAbsolute.jerk := -1.0;
   // cmSepaGripperAxisC.commandConfiguration.gearInAbsolute.syncDirection := 1;
   // cmSepaGripperAxisC.commandConfiguration.gearInAbsolute.ratioChangeOnTheFly := FALSE;
   // cmSepaGripperAxisC.commandConfiguration.gearInVelocity.continuousUpdate := FALSE;
   // cmSepaGripperAxisC.commandConfiguration.gearInVelocity.ratioNumerator := 1;
   // cmSepaGripperAxisC.commandConfiguration.gearInVelocity.ratioDenominator := 1;
   // cmSepaGripperAxisC.commandConfiguration.gearInVelocity.acceleration := -1.0;
   // cmSepaGripperAxisC.commandConfiguration.gearInVelocity.deceleration := -1.0;
   // cmSepaGripperAxisC.commandConfiguration.gearInVelocity.jerk := -1.0;
   // cmSepaGripperAxisC.commandConfiguration.gearInVelocity.positionControlled := FALSE;
   // cmSepaGripperAxisC.commandConfiguration.camIn.masterOffset := 0.0;
   // cmSepaGripperAxisC.commandConfiguration.camIn.slaveOffset := 0.0;
   // cmSepaGripperAxisC.commandConfiguration.camIn.masterScaling := 1.0;
   // cmSepaGripperAxisC.commandConfiguration.camIn.slaveScaling := 1.0;
   // cmSepaGripperAxisC.commandConfiguration.camIn.masterSyncPosition := 0.0;
   // cmSepaGripperAxisC.commandConfiguration.camIn.syncProfileReference := 1;
   // cmSepaGripperAxisC.commandConfiguration.camIn.masterStartDistance := 0.0;
   // cmSepaGripperAxisC.commandConfiguration.camIn.velocity := -1.0;
   // cmSepaGripperAxisC.commandConfiguration.camIn.acceleration := -1.0;
   // cmSepaGripperAxisC.commandConfiguration.camIn.deceleration := -1.0;
   // cmSepaGripperAxisC.commandConfiguration.camIn.jerk := -1.0;
   // cmSepaGripperAxisC.commandConfiguration.camIn.applicationMode := 0;
   // cmSepaGripperAxisC.commandConfiguration.camIn.syncDirection := 1;
   // cmSepaGripperAxisC.commandConfiguration.gearOutCamOut.slavePosition := 0.0;
   // cmSepaGripperAxisC.commandConfiguration.gearOutCamOut.syncProfileReference := 1;
   // cmSepaGripperAxisC.commandConfiguration.gearOutCamOut.masterStopDistance := 0.0;
   // cmSepaGripperAxisC.commandConfiguration.gearOutCamOut.deceleration := -1.0;
   // cmSepaGripperAxisC.commandConfiguration.gearOutCamOut.jerk := -1.0;
   // cmSepaGripperAxisC.commandConfiguration.gearOutCamOut.syncOutDirection := 3;
   // cmSepaGripperAxisC.commandConfiguration.gearOutCamOut.gearOutCamOutMode := -1;
   // cmSepaGripperAxisC.commandConfiguration.phasing.phaseShift := 0.0;
   // cmSepaGripperAxisC.commandConfiguration.phasing.velocity := -1.0;
   // cmSepaGripperAxisC.commandConfiguration.phasing.acceleration := -1.0;
   // cmSepaGripperAxisC.commandConfiguration.phasing.deceleration := -1.0;
   // cmSepaGripperAxisC.commandConfiguration.phasing.jerk := -1.0;
   // cmSepaGripperAxisC.commandConfiguration.phasing.profileReference := 0;
   // cmSepaGripperAxisC.commandConfiguration.phasing.phasingDistance := 0.0;
   // cmSepaGripperAxisC.commandConfiguration.phasing.startPosition := 0.0;
   // cmSepaGripperAxisC.commandConfiguration.phasing.direction := 3;
   // cmSepaGripperAxisC.commandConfiguration.phasing.phaseAbsolute := TRUE;
   // cmSepaGripperAxisC.commandConfiguration.phasing.phaseShiftChangeOnTheFly := FALSE;
   // cmSepaGripperAxisC.commandConfiguration.offset.offset := 0.0;
   // cmSepaGripperAxisC.commandConfiguration.offset.profileReference := 1;
   // cmSepaGripperAxisC.commandConfiguration.offset.offsetDistance := 0.0;
   // cmSepaGripperAxisC.commandConfiguration.offset.startPosition := 0.0;
   // cmSepaGripperAxisC.commandConfiguration.offset.direction := 3;
   // cmSepaGripperAxisC.commandConfiguration.offset.offsetAbsolute := TRUE;
   // cmSepaGripperAxisC.commandConfiguration.offset.offsetChangeOnTheFly := FALSE;
   // cmSepaGripperAxisC.commands.enableAxis := FALSE;
   // cmSepaGripperAxisC.commands.resetAxis := FALSE;
   // cmSepaGripperAxisC.commands.openBrake := FALSE;
   // cmSepaGripperAxisC.commands.jogForward := FALSE;
   // cmSepaGripperAxisC.commands.jogBackward := FALSE;
   // cmSepaGripperAxisC.commands.moveVelocity := FALSE;
   // cmSepaGripperAxisC.commands.stop := FALSE;
   // cmSepaGripperAxisC.commands.fastStop := FALSE;
   // cmSepaGripperAxisC.commands.torqueLimiting := FALSE;
   // cmSepaGripperAxisC.commands.homing := FALSE;
   // cmSepaGripperAxisC.commands.posRelative := FALSE;
   // cmSepaGripperAxisC.commands.posAbsolute := FALSE;
   // cmSepaGripperAxisC.commands.posSuperimposed := FALSE;
   // cmSepaGripperAxisC.commands.haltSuperimposed := FALSE;
   // cmSepaGripperAxisC.commands.selectSetPosition := -1;
   // cmSepaGripperAxisC.commands.reset := FALSE;
   // cmJRWinderRearAxisY.commandConfiguration.generalSettings.stopOnError := TRUE;
   // cmJRWinderRearAxisY.commandConfiguration.generalSettings.resetWithRestart := FALSE;
   // cmJRWinderRearAxisY.commandConfiguration.generalSettings.abortWaitingSyncCmd := TRUE;
   // cmJRWinderRearAxisY.commandConfiguration.power.startMode := 1;
   // cmJRWinderRearAxisY.commandConfiguration.power.stopMode := 0;
   // cmJRWinderRearAxisY.commandConfiguration.power.syncMotionSimulation := FALSE;
   // cmJRWinderRearAxisY.commandConfiguration.power.syncMotionSimulationExtendedMode := -1;
   // cmJRWinderRearAxisY.commandConfiguration.jog.velocity := 0.0;
   // cmJRWinderRearAxisY.commandConfiguration.jog.acceleration := -1.0;
   // cmJRWinderRearAxisY.commandConfiguration.jog.deceleration := -1.0;
   // cmJRWinderRearAxisY.commandConfiguration.jog.jerk := -1.0;
   // cmJRWinderRearAxisY.commandConfiguration.jog.positionControlled := TRUE;
   // cmJRWinderRearAxisY.commandConfiguration.jog.increment := 0.0;
   // cmJRWinderRearAxisY.commandConfiguration.jog.mode := 0;
   // cmJRWinderRearAxisY.commandConfiguration.moveVelocity.velocity := 0.0;
   // cmJRWinderRearAxisY.commandConfiguration.moveVelocity.acceleration := -1.0;
   // cmJRWinderRearAxisY.commandConfiguration.moveVelocity.deceleration := -1.0;
   // cmJRWinderRearAxisY.commandConfiguration.moveVelocity.jerk := -1.0;
   // cmJRWinderRearAxisY.commandConfiguration.moveVelocity.direction := 0;
   // cmJRWinderRearAxisY.commandConfiguration.moveVelocity.positionControlled := TRUE;
   // cmJRWinderRearAxisY.commandConfiguration.moveVelocity.velocityChangeOnTheFly := FALSE;
   // cmJRWinderRearAxisY.commandConfiguration.stop.deceleration := -1.0;
   // cmJRWinderRearAxisY.commandConfiguration.stop.jerk := -1.0;
   // cmJRWinderRearAxisY.commandConfiguration.stop.abortAcceleration := FALSE;
   // cmJRWinderRearAxisY.commandConfiguration.fastStop.deceleration := -1.0;
   // cmJRWinderRearAxisY.commandConfiguration.fastStop.jerk := -1.0;
   // cmJRWinderRearAxisY.commandConfiguration.fastStop.abortAcceleration := FALSE;
   // cmJRWinderRearAxisY.commandConfiguration.fastStop.replaceStopPossible := FALSE;
   // cmJRWinderRearAxisY.commandConfiguration.torqueLimiting.limit := -1.0;
   // cmJRWinderRearAxisY.commandConfiguration.torqueLimiting.mode := 0;
   // cmJRWinderRearAxisY.commandConfiguration.homing.position := 0.0;
   // cmJRWinderRearAxisY.commandConfiguration.homing.mode := 0;
   // cmJRWinderRearAxisY.commandConfiguration.homing.sensor := 0;
   // cmJRWinderRearAxisY.commandConfiguration.homing.extendedMode := -1;
   // cmJRWinderRearAxisY.commandConfiguration.homing.extendedModeTorqueLimit := 0.0;
   // cmJRWinderRearAxisY.commandConfiguration.homing.extendedModeTargetPosition := 0.0;
   // cmJRWinderRearAxisY.commandConfiguration.posRelative.distance := 0.0;
   // cmJRWinderRearAxisY.commandConfiguration.posRelative.velocity := -1.0;
   // cmJRWinderRearAxisY.commandConfiguration.posRelative.acceleration := -1.0;
   // cmJRWinderRearAxisY.commandConfiguration.posRelative.deceleration := -1.0;
   // cmJRWinderRearAxisY.commandConfiguration.posRelative.jerk := -1.0;
   // cmJRWinderRearAxisY.commandConfiguration.posRelative.direction := 0;
   // cmJRWinderRearAxisY.commandConfiguration.posAbsolute.position := 0.0;
   // cmJRWinderRearAxisY.commandConfiguration.posAbsolute.velocity := -1.0;
   // cmJRWinderRearAxisY.commandConfiguration.posAbsolute.acceleration := -1.0;
   // cmJRWinderRearAxisY.commandConfiguration.posAbsolute.deceleration := -1.0;
   // cmJRWinderRearAxisY.commandConfiguration.posAbsolute.jerk := -1.0;
   // cmJRWinderRearAxisY.commandConfiguration.posAbsolute.direction := 1;
   // cmJRWinderRearAxisY.commandConfiguration.posAbsolute.positionChangeOnTheFly := FALSE;
   // cmJRWinderRearAxisY.commandConfiguration.posAbsolute.velocityChangeOnTheFly := FALSE;
   // cmJRWinderRearAxisY.commandConfiguration.posSuperimposed.distance := 0.0;
   // cmJRWinderRearAxisY.commandConfiguration.posSuperimposed.velocityDiff := -1.0;
   // cmJRWinderRearAxisY.commandConfiguration.posSuperimposed.acceleration := -1.0;
   // cmJRWinderRearAxisY.commandConfiguration.posSuperimposed.deceleration := -1.0;
   // cmJRWinderRearAxisY.commandConfiguration.posSuperimposed.jerk := -1.0;
   // cmJRWinderRearAxisY.commandConfiguration.posSuperimposed.direction := 0;
   // cmJRWinderRearAxisY.commandConfiguration.haltSuperimposed.deceleration := -1.0;
   // cmJRWinderRearAxisY.commandConfiguration.haltSuperimposed.jerk := -1.0;
   // cmJRWinderRearAxisY.commandConfiguration.haltSuperimposed.abortAcceleration := FALSE;
   // cmJRWinderRearAxisY.commandConfiguration.gearInRelative.ratioNumerator := 1;
   // cmJRWinderRearAxisY.commandConfiguration.gearInRelative.ratioDenominator := 1;
   // cmJRWinderRearAxisY.commandConfiguration.gearInRelative.acceleration := -1.0;
   // cmJRWinderRearAxisY.commandConfiguration.gearInRelative.deceleration := -1.0;
   // cmJRWinderRearAxisY.commandConfiguration.gearInRelative.jerk := -1.0;
   // cmJRWinderRearAxisY.commandConfiguration.gearInRelative.ratioChangeOnTheFly := FALSE;
   // cmJRWinderRearAxisY.commandConfiguration.gearInAbsolute.ratioNumerator := 1;
   // cmJRWinderRearAxisY.commandConfiguration.gearInAbsolute.ratioDenominator := 1;
   // cmJRWinderRearAxisY.commandConfiguration.gearInAbsolute.masterSyncPosition := 0.0;
   // cmJRWinderRearAxisY.commandConfiguration.gearInAbsolute.slaveSyncPosition := 0.0;
   // cmJRWinderRearAxisY.commandConfiguration.gearInAbsolute.syncProfileReference := 1;
   // cmJRWinderRearAxisY.commandConfiguration.gearInAbsolute.masterStartDistance := 0.0;
   // cmJRWinderRearAxisY.commandConfiguration.gearInAbsolute.velocity := -1.0;
   // cmJRWinderRearAxisY.commandConfiguration.gearInAbsolute.acceleration := -1.0;
   // cmJRWinderRearAxisY.commandConfiguration.gearInAbsolute.deceleration := -1.0;
   // cmJRWinderRearAxisY.commandConfiguration.gearInAbsolute.jerk := -1.0;
   // cmJRWinderRearAxisY.commandConfiguration.gearInAbsolute.syncDirection := 1;
   // cmJRWinderRearAxisY.commandConfiguration.gearInAbsolute.ratioChangeOnTheFly := FALSE;
   // cmJRWinderRearAxisY.commandConfiguration.gearInVelocity.continuousUpdate := FALSE;
   // cmJRWinderRearAxisY.commandConfiguration.gearInVelocity.ratioNumerator := 1;
   // cmJRWinderRearAxisY.commandConfiguration.gearInVelocity.ratioDenominator := 1;
   // cmJRWinderRearAxisY.commandConfiguration.gearInVelocity.acceleration := -1.0;
   // cmJRWinderRearAxisY.commandConfiguration.gearInVelocity.deceleration := -1.0;
   // cmJRWinderRearAxisY.commandConfiguration.gearInVelocity.jerk := -1.0;
   // cmJRWinderRearAxisY.commandConfiguration.gearInVelocity.positionControlled := FALSE;
   // cmJRWinderRearAxisY.commandConfiguration.camIn.masterOffset := 0.0;
   // cmJRWinderRearAxisY.commandConfiguration.camIn.slaveOffset := 0.0;
   // cmJRWinderRearAxisY.commandConfiguration.camIn.masterScaling := 1.0;
   // cmJRWinderRearAxisY.commandConfiguration.camIn.slaveScaling := 1.0;
   // cmJRWinderRearAxisY.commandConfiguration.camIn.masterSyncPosition := 0.0;
   // cmJRWinderRearAxisY.commandConfiguration.camIn.syncProfileReference := 1;
   // cmJRWinderRearAxisY.commandConfiguration.camIn.masterStartDistance := 0.0;
   // cmJRWinderRearAxisY.commandConfiguration.camIn.velocity := -1.0;
   // cmJRWinderRearAxisY.commandConfiguration.camIn.acceleration := -1.0;
   // cmJRWinderRearAxisY.commandConfiguration.camIn.deceleration := -1.0;
   // cmJRWinderRearAxisY.commandConfiguration.camIn.jerk := -1.0;
   // cmJRWinderRearAxisY.commandConfiguration.camIn.applicationMode := 0;
   // cmJRWinderRearAxisY.commandConfiguration.camIn.syncDirection := 1;
   // cmJRWinderRearAxisY.commandConfiguration.gearOutCamOut.slavePosition := 0.0;
   // cmJRWinderRearAxisY.commandConfiguration.gearOutCamOut.syncProfileReference := 1;
   // cmJRWinderRearAxisY.commandConfiguration.gearOutCamOut.masterStopDistance := 0.0;
   // cmJRWinderRearAxisY.commandConfiguration.gearOutCamOut.deceleration := -1.0;
   // cmJRWinderRearAxisY.commandConfiguration.gearOutCamOut.jerk := -1.0;
   // cmJRWinderRearAxisY.commandConfiguration.gearOutCamOut.syncOutDirection := 3;
   // cmJRWinderRearAxisY.commandConfiguration.gearOutCamOut.gearOutCamOutMode := -1;
   // cmJRWinderRearAxisY.commandConfiguration.phasing.phaseShift := 0.0;
   // cmJRWinderRearAxisY.commandConfiguration.phasing.velocity := -1.0;
   // cmJRWinderRearAxisY.commandConfiguration.phasing.acceleration := -1.0;
   // cmJRWinderRearAxisY.commandConfiguration.phasing.deceleration := -1.0;
   // cmJRWinderRearAxisY.commandConfiguration.phasing.jerk := -1.0;
   // cmJRWinderRearAxisY.commandConfiguration.phasing.profileReference := 0;
   // cmJRWinderRearAxisY.commandConfiguration.phasing.phasingDistance := 0.0;
   // cmJRWinderRearAxisY.commandConfiguration.phasing.startPosition := 0.0;
   // cmJRWinderRearAxisY.commandConfiguration.phasing.direction := 3;
   // cmJRWinderRearAxisY.commandConfiguration.phasing.phaseAbsolute := TRUE;
   // cmJRWinderRearAxisY.commandConfiguration.phasing.phaseShiftChangeOnTheFly := FALSE;
   // cmJRWinderRearAxisY.commandConfiguration.offset.offset := 0.0;
   // cmJRWinderRearAxisY.commandConfiguration.offset.profileReference := 1;
   // cmJRWinderRearAxisY.commandConfiguration.offset.offsetDistance := 0.0;
   // cmJRWinderRearAxisY.commandConfiguration.offset.startPosition := 0.0;
   // cmJRWinderRearAxisY.commandConfiguration.offset.direction := 3;
   // cmJRWinderRearAxisY.commandConfiguration.offset.offsetAbsolute := TRUE;
   // cmJRWinderRearAxisY.commandConfiguration.offset.offsetChangeOnTheFly := FALSE;
   // cmJRWinderRearAxisY.monitoring.valid := FALSE;
   // cmJRWinderRearAxisY.monitoring.busy := TRUE;
   // cmJRWinderRearAxisY.monitoring.error := TRUE;
   // cmJRWinderRearAxisY.monitoring.status := 16#8600;
   // cmJRWinderRearAxisY.monitoring.subfunctionStatus := 16#8001;
   // cmJRWinderRearAxisY.monitoring.axisEnabled := FALSE;
   // cmJRWinderRearAxisY.monitoring.resetActive := FALSE;
   // cmJRWinderRearAxisY.monitoring.inVelocity := FALSE;
   // cmJRWinderRearAxisY.monitoring.inLimitation := FALSE;
   // cmJRWinderRearAxisY.monitoring.inClamping := FALSE;
   // cmJRWinderRearAxisY.monitoring.startSync := FALSE;
   // cmJRWinderRearAxisY.monitoring.inSync := FALSE;
   // cmJRWinderRearAxisY.monitoring.inSimulation := FALSE;
   // cmJRWinderRearAxisY.monitoring.jogSelected := FALSE;
   // cmJRWinderRearAxisY.monitoring.moveVelocitySelected := FALSE;
   // cmJRWinderRearAxisY.monitoring.stopSelected := FALSE;
   // cmJRWinderRearAxisY.monitoring.fastStopSelected := FALSE;
   // cmJRWinderRearAxisY.monitoring.torqueLimitingSelected := FALSE;
   // cmJRWinderRearAxisY.monitoring.homingSelected := FALSE;
   // cmJRWinderRearAxisY.monitoring.posRelativeSelected := FALSE;
   // cmJRWinderRearAxisY.monitoring.posAbsoluteSelected := FALSE;
   // cmJRWinderRearAxisY.monitoring.posSuperimposedSelected := FALSE;
   // cmJRWinderRearAxisY.monitoring.haltSuperimposedSelected := FALSE;
   // cmJRWinderRearAxisY.monitoring.commandBusy := FALSE;
   // cmJRWinderRearAxisY.monitoring.commandDone := FALSE;
   // cmJRWinderRearAxisY.monitoring.commandAborted := FALSE;
   // cmJRWinderRearAxisY.monitoring.homingCommandBusy := FALSE;
   // cmJRWinderRearAxisY.monitoring.homingCommandDone := FALSE;
   // cmJRWinderRearAxisY.monitoring.homingCommandAborted := FALSE;
   // cmJRWinderRearAxisY.monitoring.superimposedBusy := FALSE;
   // cmJRWinderRearAxisY.monitoring.superimposedDone := FALSE;
   // cmJRWinderRearAxisY.monitoring.superimposedAborted := FALSE;
   // cmJRWinderRearAxisY.monitoring.actualPosition := -17.994;
   // cmJRWinderRearAxisY.monitoring.actualSpeed := 0.0;
   // cmJRWinderRearAxisY.monitoring.speedUnit := 1062;
   // cmJRWinderRearAxisY.monitoring.positionUnit := 1013;
   // cmJRWinderRearAxisY.monitoring.axisType := 1;
   // cmJRWinderRearAxisY.monitoring.interlockGeneralOut := TRUE;
   // cmJRWinderRearAxisY.monitoring.interlockJogForwardOut := TRUE;
   // cmJRWinderRearAxisY.monitoring.interlockJogBackwardOut := TRUE;
   // cmJRWinderFrontAxisY.commandConfiguration.power.startMode := 1;
   // cmJRWinderFrontAxisY.commandConfiguration.power.stopMode := 0;
   // cmJRWinderFrontAxisY.commandConfiguration.power.syncMotionSimulation := FALSE;
   // cmJRWinderFrontAxisY.commandConfiguration.power.syncMotionSimulationExtendedMode := -1;
   // cmJRWinderFrontAxisY.commandConfiguration.jog.velocity := 0.0;
   // cmJRWinderFrontAxisY.commandConfiguration.jog.acceleration := -1.0;
   // cmJRWinderFrontAxisY.commandConfiguration.jog.deceleration := -1.0;
   // cmJRWinderFrontAxisY.commandConfiguration.jog.jerk := -1.0;
   // cmJRWinderFrontAxisY.commandConfiguration.jog.positionControlled := TRUE;
   // cmJRWinderFrontAxisY.commandConfiguration.jog.increment := 0.0;
   // cmJRWinderFrontAxisY.commandConfiguration.jog.mode := 0;
   // cmJRWinderFrontAxisY.commandConfiguration.moveVelocity.velocity := 0.0;
   // cmJRWinderFrontAxisY.commandConfiguration.moveVelocity.acceleration := -1.0;
   // cmJRWinderFrontAxisY.commandConfiguration.moveVelocity.deceleration := -1.0;
   // cmJRWinderFrontAxisY.commandConfiguration.moveVelocity.jerk := -1.0;
   // cmJRWinderFrontAxisY.commandConfiguration.moveVelocity.direction := 0;
   // cmJRWinderFrontAxisY.commandConfiguration.moveVelocity.positionControlled := TRUE;
   // cmJRWinderFrontAxisY.commandConfiguration.moveVelocity.velocityChangeOnTheFly := FALSE;
   // cmJRWinderFrontAxisY.commandConfiguration.stop.deceleration := -1.0;
   // cmJRWinderFrontAxisY.commandConfiguration.stop.jerk := -1.0;
   // cmJRWinderFrontAxisY.commandConfiguration.stop.abortAcceleration := FALSE;
   // cmJRWinderFrontAxisY.commandConfiguration.fastStop.deceleration := -1.0;
   // cmJRWinderFrontAxisY.commandConfiguration.fastStop.jerk := -1.0;
   // cmJRWinderFrontAxisY.commandConfiguration.fastStop.abortAcceleration := FALSE;
   // cmJRWinderFrontAxisY.commandConfiguration.fastStop.replaceStopPossible := FALSE;
   // cmJRWinderFrontAxisY.commandConfiguration.torqueLimiting.limit := -1.0;
   // cmJRWinderFrontAxisY.commandConfiguration.torqueLimiting.mode := 0;
   // cmJRWinderFrontAxisY.commandConfiguration.homing.position := 0.0;
   // cmJRWinderFrontAxisY.commandConfiguration.homing.mode := 0;
   // cmJRWinderFrontAxisY.commandConfiguration.homing.sensor := 0;
   // cmJRWinderFrontAxisY.commandConfiguration.homing.extendedMode := -1;
   // cmJRWinderFrontAxisY.commandConfiguration.homing.extendedModeTorqueLimit := 0.0;
   // cmJRWinderFrontAxisY.commandConfiguration.homing.extendedModeTargetPosition := 0.0;
   // cmJRWinderFrontAxisY.commandConfiguration.posRelative.distance := 0.0;
   // cmJRWinderFrontAxisY.commandConfiguration.posRelative.velocity := -1.0;
   // cmJRWinderFrontAxisY.commandConfiguration.posRelative.acceleration := -1.0;
   // cmJRWinderFrontAxisY.commandConfiguration.posRelative.deceleration := -1.0;
   // cmJRWinderFrontAxisY.commandConfiguration.posRelative.jerk := -1.0;
   // cmJRWinderFrontAxisY.commandConfiguration.posRelative.direction := 0;
   // cmJRWinderFrontAxisY.commandConfiguration.posAbsolute.position := 0.0;
   // cmJRWinderFrontAxisY.commandConfiguration.posAbsolute.velocity := -1.0;
   // cmJRWinderFrontAxisY.commandConfiguration.posAbsolute.acceleration := -1.0;
   // cmJRWinderFrontAxisY.commandConfiguration.posAbsolute.deceleration := -1.0;
   // cmJRWinderFrontAxisY.commandConfiguration.posAbsolute.jerk := -1.0;
   // cmJRWinderFrontAxisY.commandConfiguration.posAbsolute.direction := 1;
   // cmJRWinderFrontAxisY.commandConfiguration.posAbsolute.positionChangeOnTheFly := FALSE;
   // cmJRWinderFrontAxisY.commandConfiguration.posAbsolute.velocityChangeOnTheFly := FALSE;
   // cmJRWinderFrontAxisY.commandConfiguration.posSuperimposed.distance := 0.0;
   // cmJRWinderFrontAxisY.commandConfiguration.posSuperimposed.velocityDiff := -1.0;
   // cmJRWinderFrontAxisY.commandConfiguration.posSuperimposed.acceleration := -1.0;
   // cmJRWinderFrontAxisY.commandConfiguration.posSuperimposed.deceleration := -1.0;
   // cmJRWinderFrontAxisY.commandConfiguration.posSuperimposed.jerk := -1.0;
   // cmJRWinderFrontAxisY.commandConfiguration.posSuperimposed.direction := 0;
   // cmJRWinderFrontAxisY.commandConfiguration.haltSuperimposed.deceleration := -1.0;
   // cmJRWinderFrontAxisY.commandConfiguration.haltSuperimposed.jerk := -1.0;
   // cmJRWinderFrontAxisY.commandConfiguration.haltSuperimposed.abortAcceleration := FALSE;
   // cmJRWinderFrontAxisY.commandConfiguration.gearInRelative.ratioNumerator := 1;
   // cmJRWinderFrontAxisY.commandConfiguration.gearInRelative.ratioDenominator := 1;
   // cmJRWinderFrontAxisY.commandConfiguration.gearInRelative.acceleration := -1.0;
   // cmJRWinderFrontAxisY.commandConfiguration.gearInRelative.deceleration := -1.0;
   // cmJRWinderFrontAxisY.commandConfiguration.gearInRelative.jerk := -1.0;
   // cmJRWinderFrontAxisY.commandConfiguration.gearInRelative.ratioChangeOnTheFly := FALSE;
   // cmJRWinderFrontAxisY.commandConfiguration.gearInAbsolute.ratioNumerator := 1;
   // cmJRWinderFrontAxisY.commandConfiguration.gearInAbsolute.ratioDenominator := 1;
   // cmJRWinderFrontAxisY.commandConfiguration.gearInAbsolute.masterSyncPosition := 0.0;
   // cmJRWinderFrontAxisY.commandConfiguration.gearInAbsolute.slaveSyncPosition := 0.0;
   // cmJRWinderFrontAxisY.commandConfiguration.gearInAbsolute.syncProfileReference := 1;
   // cmJRWinderFrontAxisY.commandConfiguration.gearInAbsolute.masterStartDistance := 0.0;
   // cmJRWinderFrontAxisY.commandConfiguration.gearInAbsolute.velocity := -1.0;
   // cmJRWinderFrontAxisY.commandConfiguration.gearInAbsolute.acceleration := -1.0;
   // cmJRWinderFrontAxisY.commandConfiguration.gearInAbsolute.deceleration := -1.0;
   // cmJRWinderFrontAxisY.commandConfiguration.gearInAbsolute.jerk := -1.0;
   // cmJRWinderFrontAxisY.commandConfiguration.gearInAbsolute.syncDirection := 1;
   // cmJRWinderFrontAxisY.commandConfiguration.gearInAbsolute.ratioChangeOnTheFly := FALSE;
   // cmJRWinderFrontAxisY.commandConfiguration.gearInVelocity.continuousUpdate := FALSE;
   // cmJRWinderFrontAxisY.commandConfiguration.gearInVelocity.ratioNumerator := 1;
   // cmJRWinderFrontAxisY.commandConfiguration.gearInVelocity.ratioDenominator := 1;
   // cmJRWinderFrontAxisY.commandConfiguration.gearInVelocity.acceleration := -1.0;
   // cmJRWinderFrontAxisY.commandConfiguration.gearInVelocity.deceleration := -1.0;
   // cmJRWinderFrontAxisY.commandConfiguration.gearInVelocity.jerk := -1.0;
   // cmJRWinderFrontAxisY.commandConfiguration.gearInVelocity.positionControlled := FALSE;
   // cmJRWinderFrontAxisY.commandConfiguration.camIn.masterOffset := 0.0;
   // cmJRWinderFrontAxisY.commandConfiguration.camIn.slaveOffset := 0.0;
   // cmJRWinderFrontAxisY.commandConfiguration.camIn.masterScaling := 1.0;
   // cmJRWinderFrontAxisY.commandConfiguration.camIn.slaveScaling := 1.0;
   // cmJRWinderFrontAxisY.commandConfiguration.camIn.masterSyncPosition := 0.0;
   // cmJRWinderFrontAxisY.commandConfiguration.camIn.syncProfileReference := 1;
   // cmJRWinderFrontAxisY.commandConfiguration.camIn.masterStartDistance := 0.0;
   // cmJRWinderFrontAxisY.commandConfiguration.camIn.velocity := -1.0;
   // cmJRWinderFrontAxisY.commandConfiguration.camIn.acceleration := -1.0;
   // cmJRWinderFrontAxisY.commandConfiguration.camIn.deceleration := -1.0;
   // cmJRWinderFrontAxisY.commandConfiguration.camIn.jerk := -1.0;
   // cmJRWinderFrontAxisY.commandConfiguration.camIn.applicationMode := 0;
   // cmJRWinderFrontAxisY.commandConfiguration.camIn.syncDirection := 1;
   // cmJRWinderFrontAxisY.commandConfiguration.gearOutCamOut.slavePosition := 0.0;
   // cmJRWinderFrontAxisY.commandConfiguration.gearOutCamOut.syncProfileReference := 1;
   // cmJRWinderFrontAxisY.commandConfiguration.gearOutCamOut.masterStopDistance := 0.0;
   // cmJRWinderFrontAxisY.commandConfiguration.gearOutCamOut.deceleration := -1.0;
   // cmJRWinderFrontAxisY.commandConfiguration.gearOutCamOut.jerk := -1.0;
   // cmJRWinderFrontAxisY.commandConfiguration.gearOutCamOut.syncOutDirection := 3;
   // cmJRWinderFrontAxisY.commandConfiguration.gearOutCamOut.gearOutCamOutMode := -1;
   // cmJRWinderFrontAxisY.commandConfiguration.phasing.phaseShift := 0.0;
   // cmJRWinderFrontAxisY.commandConfiguration.phasing.velocity := -1.0;
   // cmJRWinderFrontAxisY.commandConfiguration.phasing.acceleration := -1.0;
   // cmJRWinderFrontAxisY.commandConfiguration.phasing.deceleration := -1.0;
   // cmJRWinderFrontAxisY.commandConfiguration.phasing.jerk := -1.0;
   // cmJRWinderFrontAxisY.commandConfiguration.phasing.profileReference := 0;
   // cmJRWinderFrontAxisY.commandConfiguration.phasing.phasingDistance := 0.0;
   // cmJRWinderFrontAxisY.commandConfiguration.phasing.startPosition := 0.0;
   // cmJRWinderFrontAxisY.commandConfiguration.phasing.direction := 3;
   // cmJRWinderFrontAxisY.commandConfiguration.phasing.phaseAbsolute := TRUE;
   // cmJRWinderFrontAxisY.commandConfiguration.phasing.phaseShiftChangeOnTheFly := FALSE;
   // cmJRWinderFrontAxisY.commandConfiguration.offset.offset := 0.0;
   // cmJRWinderFrontAxisY.commandConfiguration.offset.profileReference := 1;
   // cmJRWinderFrontAxisY.commandConfiguration.offset.offsetDistance := 0.0;
   // cmJRWinderFrontAxisY.commandConfiguration.offset.startPosition := 0.0;
   // cmJRWinderFrontAxisY.commandConfiguration.offset.direction := 3;
   // cmJRWinderFrontAxisY.commandConfiguration.offset.offsetAbsolute := TRUE;
   // cmJRWinderFrontAxisY.commandConfiguration.offset.offsetChangeOnTheFly := FALSE;
END_TYPE
